PROGRAM InterfaceLink
VAR
	iResult					: INT;
	iLoopFBAnalogIn			: INT;
	iLoopFBSensor			: INT;
	iLoopFBValveSensor		: INT;
	iLoopFBDigCtrl			: INT;
	iLoopFBValveCtrl		: INT;
	uiLoopDMXCtrlI			: UINT;
	uiLoopDMXCtrlII			: UINT;
	uiLoopDebouncePNPI		: UINT;
	uiLoopDebounceNPNI		: UINT;
END_VAR

//Call all the I/O Function Blocks continuously; link to array-structs with every call;
(*
FOR iLoopFBAnalogIn := 0 TO gc.usiMaxNrOfAnalogIn BY 1 DO
	gFB.arrFB_AnalogInput[iLoopFBAnalogIn](I:=gast_AnalogInput[iLoopFBAnalogIn].I, IQ:=gast_AnalogInput[iLoopFBAnalogIn].IQ, Q=>gast_AnalogInput[iLoopFBAnalogIn].Q);
END_FOR

FOR iLoopFBSensor := 0 TO gc.usiMaxNrOfSensor BY 1 DO
	gFB.arrFB_Sensor[iLoopFBSensor](I:=gast_SensorInput[iLoopFBSensor].I, IQ:=gast_SensorInput[iLoopFBSensor].IQ, Q=>gast_SensorInput[iLoopFBSensor].Q);
END_FOR

FOR iLoopFBValveSensor := 0 TO (2*gc.usiMaxNrOfValveCtrl) BY 1 DO
	gFB.arrFB_Sensor[iLoopFBValveSensor](I:=gast_ValveSensorInput[iLoopFBValveSensor].I, IQ:=gast_ValveSensorInput[iLoopFBValveSensor].IQ, Q=>gast_ValveSensorInput[iLoopFBValveSensor].Q);
END_FOR

FOR iLoopFBDigCtrl := 0 TO gc.usiMaxNrOfSensor BY 1 DO
	gFB.arrFB_DigCtrl[iLoopFBDigCtrl](I:=gast_DigCtrlOutput[iLoopFBDigCtrl].I, IQ:=gast_DigCtrlOutput[iLoopFBDigCtrl].IQ, Q=>gast_DigCtrlOutput[iLoopFBDigCtrl].Q);
END_FOR

FOR iLoopFBValveCtrl := 0 TO gc.usiMaxNrOfValveCtrl BY 1 DO
	gFB.arrFB_ValveCtrl[iLoopFBValveCtrl](I:=gast_ValveCtrlOutput[iLoopFBValveCtrl].I, IQ:=gast_ValveCtrlOutput[iLoopFBValveCtrl].IQ, Q=>gast_ValveCtrlOutput[iLoopFBValveCtrl].Q);
END_FOR
*)
FOR uiLoopDMXCtrlI := 0 TO gc.uiMaxNrOfDMXChannel BY 1 DO
	gFB.arrFB_DMX[uiLoopDMXCtrlI](I:=g_ast.DMX[uiLoopDMXCtrlI].I, IQ:=g_ast.DMX[uiLoopDMXCtrlI].IQ, Q=>g_ast.DMX[uiLoopDMXCtrlI].Q);
END_FOR

//Expose an array of bytes that can be ultimately 'multi-linked' to hardware
FOR uiLoopDMXCtrlII := 0 TO gc.uiMaxNrOfDMXChannel BY 1 DO
	g_ast.DMXPhysOut[uiLoopDMXCtrlII]	:= g_ast.DMX[uiLoopDMXCtrlII].Q.byStatValue;
END_FOR

//Debounce PNP
FOR uiLoopDebouncePNPI	:= 0 TO gc.uiMaxNrDMXTestCh BY 1 DO
	gFB.arrFB_DebouncePNP[uiLoopDebouncePNPI](I:=g_ast.arrFBIntPNP[uiLoopDebouncePNPI].I, IQ:=g_ast.arrFBIntPNP[uiLoopDebouncePNPI].IQ, Q=>g_ast.arrFBIntPNP[uiLoopDebouncePNPI].Q);
END_FOR

//Debounce NPN
FOR uiLoopDebounceNPNI	:= 0 TO gc.uiMaxNrDMXTestCh BY 1 DO
	gFB.arrFB_DebounceNPN[uiLoopDebounceNPNI](I:=g_ast.arrFBIntNPN[uiLoopDebounceNPNI].I, IQ:=g_ast.arrFBIntNPN[uiLoopDebounceNPNI].IQ, Q=>g_ast.arrFBIntNPN[uiLoopDebounceNPNI].Q);
END_FOR

END_PROGRAM

(* stored: Version 1.1.0.1, ProductVersion 3.1.4024.6
   POU InterfaceLink: Id {e5515fc8-d968-4a6f-8e7a-8841024cd466}, SpecialFunc None *)
